FUNCTION_BLOCK SU2 (* Basic FB with empty ECC *)
  (* Standard: 61499-2 *)
  (* Version 1.0, 0000-00-00, 0 *)
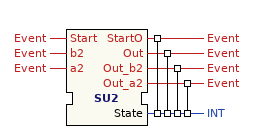
  EVENT_INPUT
    Start;
    b2;
    a2;
  END_EVENT
  EVENT_OUTPUT
    StartO WITH State;
    Out WITH State;
    Out_b2 WITH State;
    Out_a2 WITH State;
  END_EVENT
  VAR_OUTPUT
    State : INT := 1;
  END_VAR
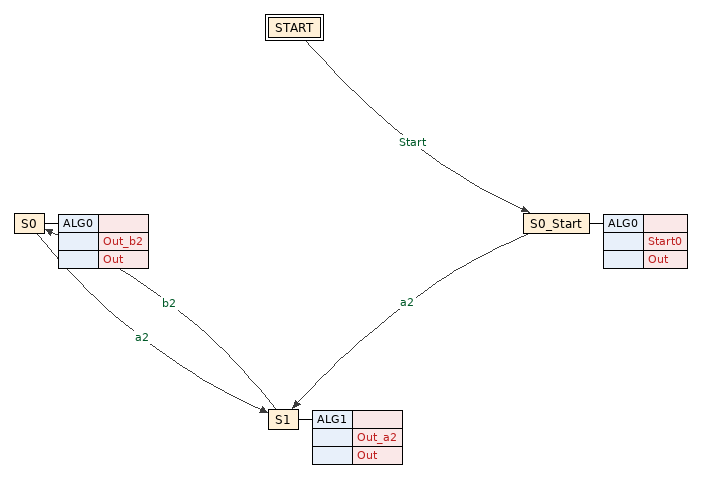
  EC_STATES
    START; (* Initial State *)
    S0_Start : ALG0, -> Start0, -> Out;
    S1 : ALG1, -> Out_a2, -> Out;
    S0 : ALG0, -> Out_b2, -> Out;
  END_STATES
  EC_TRANSITIONS
    START TO S0_Start := Start;
    S0_Start TO S1 := a2;
    S0 TO S1 := a2;
    S1 TO S0 := b2;
  END_TRANSITIONS
  ALGORITHM ALG1 IN ST:
State:=1;
  END_ALGORITHM
  ALGORITHM ALG0 IN ST:
State:=0;
  END_ALGORITHM
END_FUNCTION_BLOCK
